FUNCTION_BLOCK Phase_HMI (* Service Interface Function Block Type *)
  (* Standard: 61499-2 *)
  (* Version 0.0, 6/4/2026, Schneider Electric, template *)
  PACKAGE SE.Nereda;
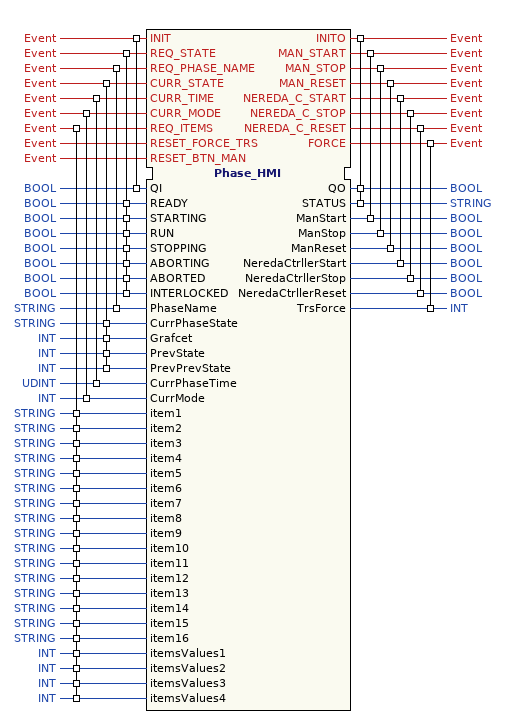
  EVENT_INPUT
    INIT WITH QI;
    REQ_STATE WITH STARTING, RUN, STOPPING, ABORTING, ABORTED, INTERLOCKED, READY;
    REQ_PHASE_NAME WITH PhaseName;
    CURR_STATE WITH CurrPhaseState, Grafcet, PrevState, PrevPrevState;
    CURR_TIME WITH CurrPhaseTime;
    CURR_MODE WITH CurrMode;
    REQ_ITEMS WITH item1, item2, item3, item4, item5, item6, item7, item8, itemsValues1, itemsValues2, item9, item10, item11, item12, item13, item14, item15, item16, itemsValues3, itemsValues4;
    RESET_FORCE_TRS;
    RESET_BTN_MAN;
  END_EVENT
  EVENT_OUTPUT
    INITO WITH QO, STATUS;
    MAN_START WITH ManStart;
    MAN_STOP WITH ManStop;
    MAN_RESET WITH ManReset;
    NEREDA_C_START WITH NeredaCtrllerStart;
    NEREDA_C_STOP WITH NeredaCtrllerStop;
    NEREDA_C_RESET WITH NeredaCtrllerReset;
    FORCE WITH TrsForce;
  END_EVENT
  VAR_INPUT
    QI : BOOL;
    READY : BOOL;
    STARTING : BOOL;
    RUN : BOOL;
    STOPPING : BOOL;
    ABORTING : BOOL;
    ABORTED : BOOL;
    INTERLOCKED : BOOL;
    PhaseName : STRING;
    CurrPhaseState : STRING;
    Grafcet : INT;
    PrevState : INT;
    PrevPrevState : INT;
    CurrPhaseTime : UDINT;
    CurrMode : INT;
    item1 : STRING;
    item2 : STRING;
    item3 : STRING;
    item4 : STRING;
    item5 : STRING;
    item6 : STRING;
    item7 : STRING;
    item8 : STRING;
    item9 : STRING;
    item10 : STRING;
    item11 : STRING;
    item12 : STRING;
    item13 : STRING;
    item14 : STRING;
    item15 : STRING;
    item16 : STRING;
    itemsValues1 : INT;
    itemsValues2 : INT;
    itemsValues3 : INT;
    itemsValues4 : INT;
  END_VAR
  VAR_OUTPUT
    QO : BOOL; (* Event Output Qualifier *)
    STATUS : STRING; (* Service Status *)
    ManStart : BOOL;
    ManStop : BOOL;
    ManReset : BOOL;
    NeredaCtrllerStart : BOOL;
    NeredaCtrllerStop : BOOL;
    NeredaCtrllerReset : BOOL;
    TrsForce : INT;
  END_VAR
  SERVICE /
    SEQUENCE 
    END_SEQUENCE
  END_SERVICE
END_FUNCTION_BLOCK
